{attribute 'GeneratedUsingTerminal: EL6861-0000-0016'}
{attribute addProperty BoxType "EL6861-0000-0016"}
{attribute addProperty Id "COM_TxPDO_Map_InputsAT %I*COM_TxPDO_Map_Inputs_93BAD1D7137COM_RxPDO_MapAT %Q*COM_RxPDO_Map_01DE24DC133WcStateAT %I*WcState_9091E0EB2InfoDataAT %I*InfoData_94A18F5E2"}
{attribute addProperty CRC "1128006240"}
{attribute addProperty Size "274"}
TYPE EL6861_433C0260 EXTENDS EtcSlaveTerminalBase_947E5A46 :
STRUCT
	{attribute addProperty Name "COM_TxPDO_Map_Inputs"}
	COM_TxPDO_Map_Inputs : COM_TxPDO_Map_Inputs_93BAD1D7;
	{attribute addProperty Name "COM_RxPDO_Map"}
	COM_RxPDO_Map : COM_RxPDO_Map_01DE24DC;
	{attribute addProperty Name "WcState"}
	WcState : WcState_9091E0EB;
	{attribute addProperty Name "InfoData"}
	InfoData : InfoData_94A18F5E;
END_STRUCT
END_TYPE

(* stored: Version 1.2.0.0, ProductVersion 3.1.4024.9
   DUT EL6861_433C0260: Id {0e80168b-585c-4861-ae10-805d297e1d0e} *)
